// TIA Portal V20 export
DATA_BLOCK "SP501"   // DB341
// stored: MemoryReserve 100
   VAR
      "CONTROL DC POWER TRIPPED E156CB" : Bool := TRUE;
      "SAFETY DC POWER TRIPPED E218CB" : Bool := TRUE;
      "CLASS 2 SMPS POWER TRIPPED E308CB" : Bool := TRUE;
      "CLASS 2 SMPS MONITORING E310PWS" : Bool := TRUE;
      "ET200ECO PN-1 POWER TRIPPED E324CB" : Bool := TRUE;
      "ET200ECO PN-2 POWER TRIPPED E328CB" : Bool := TRUE;
      "ET200ECO PN-3 POWER TRIPPED E332CB" : Bool := TRUE;
      "ET200ECO PN-4 POWER TRIPPED E336CB" : Bool := TRUE;
      "SEPA UW IONIZER TOP MAINTERNANCE DETECTION" : Bool := FALSE;
      "SEPA UW IONIZER TOP ERROR" : Bool := TRUE;
      SPARE : Bool := FALSE;
      SPARE_1 : Bool := FALSE;
      "SEPA UW IONIZER BOTTOM MAINTERNANCE DETECTION" : Bool := FALSE;
      "SEPA UW IONIZER BOTTOM ERROR" : Bool := TRUE;
      SPARE_2 : Bool := FALSE;
      SPARE_3 : Bool := FALSE;
   END_VAR
BEGIN
END_DATA_BLOCK
